INTERFACE I_TempSensor EXTENDS I_ComponentBase

PROPERTY SimulatedHeatingElement : I_HeatingElement
GET
END_GET
SET
END_SET
END_PROPERTY

PROPERTY Temp : LREAL
GET
END_GET
END_PROPERTY

END_INTERFACE

(* stored: Version 1.1.0.1
   Itf I_TempSensor: Id {50c55809-fda1-447d-bc3e-8203634c9af0}
   Property SimulatedHeatingElement: Id {1d486f18-5279-4230-9146-e7fa3cd5c9d1}
   Get Get: Id {11015281-fa0b-45e2-89b0-ec25227c39ca}
   Set Set: Id {12cb8d8b-8de6-4dde-aa46-d3a5d52aa0bf}
   Property Temp: Id {ce127390-c556-41bd-a4b2-3337fb4d92d9}
   Get Get: Id {80d78f06-89c8-4b0b-bd29-caf0d50c6508} *)
